(* PLC project CoDeSys External Library Template, WAGO e!COCKPIT e!COCKPIT, author 3S - Smart Software Solutions GmbH *)
(* stored: creationDateTime 2019-10-29T12:22:40.6358606, version 3.5.5.30, modificationDateTime 2019-10-24T14:40:07.960949, organization 3S - Smart Software Solutions GmbH *)
(* Library project template with all possible element types, docu and a sample project structure *)

FUNCTION_BLOCK fbModbusDriverRTU
  VAR_INPUT
    intOdczytZapisZadanieRozmiarBufora : INT;
    arRTUParametryKomunikacji : ARRAY[1..256] OF typModbusRTUParametryKomunikacji;
  END_VAR
  VAR_IN_OUT
    arOdczytCykliczny : ARRAY[1..5000] OF typModbusOdczytCykliczny;
    arOdczytZapisZadanie : ARRAY[1..1000] OF typModbusOdczytZapisZadanie;
    arStatusKomunikacji : ARRAY[1..256] OF INT;
    intZnacznikOdczytuZapisuZadanie : INT;
  END_VAR
  VAR
    ModbusMasterRTU : FbMbMasterSerial;
    arRTUParametryKomunikacjiPoprz : ARRAY[1..256] OF typModbusRTUParametryKomunikacji;
    utZapytanie : typMBQuery;
    utZapytaniePoprz : typMBQuery;
    utOdpowiedz : typMbResponse;
    xStatusPolaczenia : BOOL;
    xBladKomunikacji : BOOL;
    typStatusKomunikacji : WagoSysErrorBase.FbResult;
    tCzasPonowienia : LTIME := LTIME#15s0ms0us0ns;
    tCzasStabilnosciKomunikacji : LTIME := LTIME#30s0ms0us0ns;  (* czas po jakim driver raportuje poprawną komunikację po jej faktycznym odzyskaniu - czas powinien być większy niż czas tCzasPonawiania *)
    xDriverWykonajKomunikacje : BOOL;  (* zmienna sygnalizujaca konicznosc wykonania zapisu/odczytu do Modbus RTU *)
    tonDriverWykonajKomunikacje : TON;  (* Opóżnienie włączenia triggera wysłania komunikatu po włączeniu drivera MODBUSa *)
    xDriverWykonajKomunikacjeTrigger : BOOL;  (* Trigger wysłania komunikatu MODBUS *)
    ftrigDriverWykonajKomunikacjeTrigger : F_TRIG;  (* Zbocze opadające triggera wysłania komunikatu *)
    arStatusKomunikacjiTimestampOstatniaProba : ARRAY[1..256] OF LTIME;
    arStatusKomunikacjiTimestampOstatniBlad : ARRAY[1..256] OF LTIME;
    negWykonaj : F_TRIG;
    intZnacznikDriveraOdczytuCyklicznego : INT := 0;
    intZnacznikDriveraOdczytuZapisuZadanie : INT := 0;
    intZnacznikOdczytuCyklicznegoReferencja : INT;
    intZnacznikOdczytuCyklicznegoPoczatek : INT;
    intZnacznikOdczytuZapisuZadanieReferencja : INT;
    intZnacznikPomocniczy : INT;
    intOdczytZadanieTablica : INT;
    intOdczytCyklicznyTablica : INT;
    intOdczytCyklicznyTablicaIlosc : INT;
    intLoop : INT;
    intLoopOverflow : INT;
    statusbledu : WagoSysErrorBase.FbResult;
    jakiezapytanie : typMBQuery;
    intDebugZnacznik : INT;  (* debug *)
    arDebugZapytanie : ARRAY[0..5000] OF typMBQuery;
    arDebugOdpowiedz : ARRAY[0..5000] OF typMbResponse;
    typDebugOdczytZapisZadanie : ARRAY[0..5000] OF typModbusOdczytZapisZadanie;
    arDebugCzas : ARRAY[0..5000] OF DT;
    inttest : DINT;
    ctuLicznikBledow : CTU;  (* Licznik błędów *)
  END_VAR

            (*			
Autor:					N/A
Prawa majątkowe: 		Solwena Sp. z o.o., 
Aktualizacje:								

Opis:					Obsługa komunikacji MODBUS
						
Aktualizacje:			2019-09-13-AWy: zmiana sposobu uruchamiania drivera MODBUSowego ModbusMasterRTU i wysyłania komunkatów.
						2019-10-18-AWy: dodanie licznika błędów
						2019-10-22-AWy: zmiana opóżnienia włączenia drivera po zakończeniu komunikacji
						
Rozwój:					Możliwe jest przyspieszenie drivera poprzez nie restartowanie po każdej komunikacji a jedynie wtedy, gdy ulegną zmianie parametry komunikacji.						
	
*)

// obsługa odczytu/zapisu danych na żądanie

IF intZnacznikDriveraOdczytuZapisuZadanie <> intZnacznikOdczytuZapisuZadanie AND NOT xDriverWykonajKomunikacje THEN
	fnTablicaKomunikatowInkrementacja(intRozmiarTablicy := intOdczytZapisZadanieRozmiarBufora, intWskaznik := intZnacznikDriveraOdczytuZapisuZadanie);
	IF arStatusKomunikacji[arOdczytZapisZadanie[intZnacznikDriveraOdczytuZapisuZadanie].bAdresUrzadzenia] = enumModbusStatus.KomunikacjaPrawidlowa THEN
		xDriverWykonajKomunikacje := TRUE;
		utZapytanie.bUnitId := arOdczytZapisZadanie[intZnacznikDriveraOdczytuZapisuZadanie].bAdresUrzadzenia;
		utZapytanie.bFunctionCode := arOdczytZapisZadanie[intZnacznikDriveraOdczytuZapisuZadanie].bFunkcja;
		utZapytanie.uiReadQuantity := 1;
		utZapytanie.uiReadAddress := arOdczytZapisZadanie[intZnacznikDriveraOdczytuZapisuZadanie].uiAdresRejestru;
		utZapytanie.uiWriteAddress := arOdczytZapisZadanie[intZnacznikDriveraOdczytuZapisuZadanie].uiAdresRejestru;
		utZapytanie.awWriteData[0] := arOdczytZapisZadanie[intZnacznikDriveraOdczytuZapisuZadanie].wWartoscDoZapisania;
		utZapytanie.uiWriteQuantity := 1;
		intOdczytZadanieTablica := intZnacznikDriveraOdczytuZapisuZadanie;
	END_IF
END_IF

// obsługa odczytu cyklicznego zmiennych zapisanych w tabeli

IF NOT xDriverWykonajKomunikacje THEN 
	
	intZnacznikOdczytuCyklicznegoReferencja := intZnacznikDriveraOdczytuCyklicznego;
	intZnacznikDriveraOdczytuCyklicznego := intZnacznikDriveraOdczytuCyklicznego + 1;
	IF arOdczytCykliczny[intZnacznikDriveraOdczytuCyklicznego].bAdresUrzadzenia = 0 THEN
		intZnacznikDriveraOdczytuCyklicznego := 1;
	END_IF

	WHILE intZnacznikOdczytuCyklicznegoReferencja <> intZnacznikDriveraOdczytuCyklicznego AND _GetLongTime() - arStatusKomunikacjiTimestampOstatniaProba[arOdczytCykliczny[intZnacznikDriveraOdczytuCyklicznego].bAdresUrzadzenia] < tCzasPonowienia AND
			_GetLongTime() - arOdczytCykliczny[intZnacznikDriveraOdczytuCyklicznego].ltZnacznikCzasuWyslania < arOdczytCykliczny[intZnacznikDriveraOdczytuCyklicznego].ltCzestotliwosc DO
		intZnacznikDriveraOdczytuCyklicznego := intZnacznikDriveraOdczytuCyklicznego + 1;
		IF arOdczytCykliczny[intZnacznikDriveraOdczytuCyklicznego].bAdresUrzadzenia = 0 THEN
			intZnacznikDriveraOdczytuCyklicznego := 1;
		END_IF
	END_WHILE

// zapis adresu startowego rejestrów do zapisu

	IF intZnacznikOdczytuCyklicznegoReferencja <> intZnacznikDriveraOdczytuCyklicznego THEN
		xDriverWykonajKomunikacje := TRUE;
		arStatusKomunikacjiTimestampOstatniaProba[arOdczytCykliczny[intZnacznikDriveraOdczytuCyklicznego].bAdresUrzadzenia] := _GetLongTime();
		utZapytanie.bUnitId := arOdczytCykliczny[intZnacznikDriveraOdczytuCyklicznego].bAdresUrzadzenia;
		utZapytanie.bFunctionCode := arOdczytCykliczny[intZnacznikDriveraOdczytuCyklicznego].bFunkcja;
		utZapytanie.uiReadAddress := arOdczytCykliczny[intZnacznikDriveraOdczytuCyklicznego].uiAdresRejestru;
		utZapytanie.uiReadQuantity := 1;
		intOdczytCyklicznyTablica := intZnacznikDriveraOdczytuCyklicznego;
		intZnacznikOdczytuCyklicznegoReferencja := intZnacznikDriveraOdczytuCyklicznego;
		intZnacznikPomocniczy := intZnacznikDriveraOdczytuCyklicznego + 1;
		IF arOdczytCykliczny[intZnacznikPomocniczy].bAdresUrzadzenia = 0 THEN
			intZnacznikPomocniczy := 1;
		END_IF

// sprawdzenie czy następne żądanie nie jest w kolejności do bieżącego jeśli tak to grupuje je w jedno zapytanie

		WHILE (arOdczytCykliczny[intZnacznikPomocniczy].uiAdresRejestru - arOdczytCykliczny[intZnacznikDriveraOdczytuCyklicznego].uiAdresRejestru = 1 AND
				arOdczytCykliczny[intZnacznikPomocniczy].bFunkcja = arOdczytCykliczny[intZnacznikDriveraOdczytuCyklicznego].bFunkcja AND
				arOdczytCykliczny[intZnacznikPomocniczy].bAdresUrzadzenia = arOdczytCykliczny[intZnacznikDriveraOdczytuCyklicznego].bAdresUrzadzenia) DO
				
			utZapytanie.uiReadQuantity := utZapytanie.uiReadQuantity + 1;
			intZnacznikDriveraOdczytuCyklicznego := intZnacznikDriveraOdczytuCyklicznego + 1;
			IF arOdczytCykliczny[intZnacznikDriveraOdczytuCyklicznego].bAdresUrzadzenia = 0 THEN
				intZnacznikDriveraOdczytuCyklicznego := 1;
			END_IF
			intZnacznikPomocniczy := intZnacznikDriveraOdczytuCyklicznego + 1;
			IF arOdczytCykliczny[intZnacznikPomocniczy].bAdresUrzadzenia = 0 THEN
				intZnacznikPomocniczy := 1;
			END_IF
		END_WHILE
		intOdczytCyklicznyTablicaIlosc := UINT_TO_INT(utZapytanie.uiReadQuantity);
	END_IF
END_IF

// driver komunikacyjny MODBUS RTU
	// Na potrzeby obsługi komunikacji w kilku prędkościach: ModbusMasterRTU jest włączany (xConnect := TRUE), wprowadzane są nowe parametry komunikacji, a następnie triggerowane jest wysłanie komunikatu
	// (xTrigger := TRUE). Następnie ModbusMasterRTU jest wyłączany (xConnect := FALSE) i algorytm zaczyna się od nowa.

ftrigDriverWykonajKomunikacjeTrigger(CLK := xDriverWykonajKomunikacjeTrigger);
IF ftrigDriverWykonajKomunikacjeTrigger.Q THEN
	xDriverWykonajKomunikacje := FALSE;
END_IF

tonDriverWykonajKomunikacje(IN := xDriverWykonajKomunikacje, PT := T#1000MS); // Opóżnienie konieczne ze względu na nieprawidłowe działanie drivera przy zbyt szybkim wysyłaniu komunikatu po włączeniu drivera
IF tonDriverWykonajKomunikacje.Q THEN
	xDriverWykonajKomunikacjeTrigger := TRUE;
END_IF		

ModbusMasterRTU(xConnect := 		xDriverWykonajKomunikacje,
				I_Port := 			arRTUParametryKomunikacji[utZapytanie.bUnitId].typNazwaPortuKomunikacyjnego , 
				eFrameType := 		arRTUParametryKomunikacji[utZapytanie.bUnitId].eTypRamki , 
				udiBaudrate := 		arRTUParametryKomunikacji[utZapytanie.bUnitId].udiPredkosc , 
				usiDataBits := 		arRTUParametryKomunikacji[utZapytanie.bUnitId].usiBityDanych , 
				eParity := 			arRTUParametryKomunikacji[utZapytanie.bUnitId].eParzystosc , 
				eStopBits := 		arRTUParametryKomunikacji[utZapytanie.bUnitId].eBityStopu , 
				eHandshake :=		arRTUParametryKomunikacji[utZapytanie.bUnitId].eHandshake , 
				ePhysical := 		arRTUParametryKomunikacji[utZapytanie.bUnitId].eDuplex , 
				tTimeOut := 		arRTUParametryKomunikacji[utZapytanie.bUnitId].tTimeout , 
 
				xTrigger := 		xDriverWykonajKomunikacjeTrigger , 
				utQuery := 			utZapytanie , 
				utResponse := 		utOdpowiedz ,
 
				xError => 			xBladKomunikacji);
				
// Licznik błędów
ctuLicznikBledow(CU := ModbusMasterRTU.xError, PV := 65535);
	
// obługa akcji po zakończeniu zadania komunikacji (zapis wartości , zapis błędu itd)
	
negWykonaj(CLK := xDriverWykonajKomunikacjeTrigger);

IF negWykonaj.Q THEN
// jeżeli był błąd komunikacji wpisz go do tablicy błędów

	IF xBladKomunikacji THEN
		arStatusKomunikacji[utZapytanie.bUnitId] := enumModbusStatus.BrakKomunikacji;
		statusbledu := ModbusMasterRTU.oStatus;
		jakiezapytanie := utZapytanie;
		arStatusKomunikacjiTimestampOstatniBlad[utZapytanie.bUnitId] := _GetLongTime();
		IF utZapytaniePoprz.bFunctionCode = 0 THEN
			utZapytaniePoprz := utZapytanie;
		END_IF
		IF arRTUParametryKomunikacjiPoprz[3].udiPredkosc = 0 THEN
			arRTUParametryKomunikacjiPoprz := arRTUParametryKomunikacji;
		END_IF
	ELSE
		IF _GetLongTime() - arStatusKomunikacjiTimestampOstatniBlad[utZapytanie.bUnitId] > tCzasStabilnosciKomunikacji AND arStatusKomunikacji[utZapytanie.bUnitId] <> enumModbusStatus.KomunikacjaPrawidlowa THEN	
			arStatusKomunikacji[utZapytanie.bUnitId] := enumModbusStatus.KomunikacjaPrawidlowa;
		END_IF

// jeżeli zapytanie było żądaniem  wysłania danych

		IF utZapytanie.bFunctionCode = enumModbusKodyFunkcji.OdczytWejscBitowych OR utZapytanie.bFunctionCode = enumModbusKodyFunkcji.OdczytWyjscBitowych OR
			utZapytanie.bFunctionCode = enumModbusKodyFunkcji.OdczytNRejestrow OR utZapytanie.bFunctionCode = enumModbusKodyFunkcji.OdczytNRejestrowWejsciowych THEN
			intZnacznikOdczytuCyklicznegoPoczatek := 0;
		
// jeżeli był wykonany rozkaz odczytu danych z cyklu "na żądanie" - DOŁOŻONO KAWAŁEK KODU DEBUGUJĄCEGO - ZATRZYMYWANIE SIĘ STEROWNIKA NA ZAREMOWANEJ LINII

			IF intOdczytZadanieTablica <> 0 THEN
				arDebugZapytanie[intDebugZnacznik] := utZapytanie;
				arDebugOdpowiedz[intDebugZnacznik] := utOdpowiedz;
				typDebugOdczytZapisZadanie[intDebugZnacznik] := arOdczytZapisZadanie[intZnacznikDriveraOdczytuZapisuZadanie];				
				arDebugCzas[intDebugZnacznik] := FuGetDateAndTime();
				fnTablicaKomunikatowInkrementacja(intRozmiarTablicy := 900, intWskaznik := intDebugZnacznik);
//				arOdczytZapisZadanie[intZnacznikDriveraOdczytuZapisuZadanie].pZmiennaDoOdczytu^ := utOdpowiedz.awData[0];
			END_IF

// jeżeli był wykonany rozkaz odczytu danych z cyklu "cykliczny"

			IF intOdczytCyklicznyTablica <> 0 THEN
				intLoopOverflow:=1;
				FOR intLoop := 1 TO intOdczytCyklicznyTablicaIlosc DO
					IF arOdczytCykliczny[intOdczytCyklicznyTablica + intLoop - 1].pZmiennaReferencyjna <> null THEN
					arOdczytCykliczny[intOdczytCyklicznyTablica + intLoop - 1].pZmiennaReferencyjna^ := utOdpowiedz.awData[intLoop - 1];
					arOdczytCykliczny[intOdczytCyklicznyTablica + intLoop - 1].ltZnacznikCzasuWyslania := _GetLongTime();
					ELSE
					arOdczytCykliczny[intLoopOverflow].pZmiennaReferencyjna^ := utOdpowiedz.awData[intLoop - 1];
					arOdczytCykliczny[intLoopOverflow].ltZnacznikCzasuWyslania := _GetLongTime();
					intLoopOverflow:=intLoopOverflow+1;
					END_IF
				END_FOR
			END_IF
		END_IF
	END_IF
	intOdczytZadanieTablica := 0;
	intOdczytCyklicznyTablica := 0;
	intOdczytCyklicznyTablicaIlosc := 0;
END_IF


          
END_FUNCTION_BLOCK
